Fanuc KAREL source: port_WDOUT.kl

PROGRAM TP
%NOLOCKGROUP
VAR
 x: BOOLEAN
BEGIN
 x = WDOUT[3]
END TP
